Omron Sysmac Studio project TicTacToe (Sysmac Studio 1.60.0.64010, StandardProject)

# Controller new_Controller_0: NJ501-1500 version 1.67
Units and slaves: Power Supply : NJ-Px3001; CPU : NJ501-1500
Task PrimaryTask (priority 4, period or condition 1000): Program0

VAR_GLOBAL CONSTANT
    Table_HMI_Mapping : ARRAY[0..2,0..2] of uint := [1, 2, 3, 4, 5, 6, 7, 8, 9];  (* Use for HMI input mapping ONYL *)
END_VAR
VAR_GLOBAL
    Game_Start : BOOL;  (* Game Start Indicator *)
    Game_ReStart : BOOL;  (* Restart BTN *)
    PlayTable : ARRAY[0..2,0..2] of uint := [9(0)];
    Game_End : BOOL;  (* Game End Indicator *)
    WINNING_PLAYER : UINT;
    Player_Click : BOOL;  (* HMI BTN Detected *)
    BTN_LOCATION : UINT;
    PLAYER_1_ON : BOOL;
    PLAYER_2_ON : BOOL;
    row : UINT;
    col : UINT;
END_VAR

PROGRAM Program0
VAR
    CLEAR_TABLE : BOOL;  (* CLEAR TABLE DATA *)
    PLAYER_1_ACTIVATE : BOOL;
    PLAYER_2_ACTIVATE : BOOL;
    SWITCH_PLAYER : BOOL;
    INST_VALUE : UINT;  (* 0 = ERROR /       1= PLAYER_1        2= PLAYER_2 *)
    CheckInput : BOOL;
    CheckInput_DONE : BOOL;
END_VAR
VAR CONSTANT
    Table_Mapping_Col : Array[0..9] of Uint := [5, 0, 1, 2, 0, 1, 2, 0, 1, 2];
    Table_Mapping_Row : Array[0..9] of Uint := [5, 3(0), 3(1), 3(2)];
END_VAR
VAR_EXTERNAL
    Game_Start : BOOL;
    Game_ReStart : BOOL;
    PlayTable : ARRAY[0..2,0..2] of uint;
    Game_End : BOOL;
    WINNING_PLAYER : UINT;
    Player_Click : BOOL;
    PLAYER_1_ON : BOOL;
    PLAYER_2_ON : BOOL;
    BTN_LOCATION : UINT;
    row : UINT;
    col : UINT;
END_VAR
VAR
    _p1 : BOOL;
    _e2 : R_TRIG;
    _p3 : BOOL;
    _e4 : R_TRIG;
    _p5 : BOOL;
    _p6 : BOOL;
    _p7 : BOOL;
    _e8 : R_TRIG;
    _e9 : R_TRIG;
    _e10 : R_TRIG;
    _p11 : BOOL;
    _e12 : R_TRIG;
    _e13 : R_TRIG;
    _e14 : R_TRIG;
    _p15 : BOOL;
    _e16 : R_TRIG;
    _e17 : R_TRIG;
    _e18 : R_TRIG;
    _p19 : BOOL;
    _e20 : R_TRIG;
    _e21 : R_TRIG;
    _e22 : R_TRIG;
    _p23 : BOOL;
    _e24 : R_TRIG;
    _e25 : R_TRIG;
    _e26 : R_TRIG;
    _p27 : BOOL;
    _e28 : R_TRIG;
    _e29 : R_TRIG;
    _e30 : R_TRIG;
    _p31 : BOOL;
    _e32 : R_TRIG;
    _e33 : R_TRIG;
    _e34 : R_TRIG;
    _p35 : BOOL;
    _e36 : R_TRIG;
    _e37 : R_TRIG;
    _e38 : R_TRIG;
    _p39 : BOOL;
END_VAR

(* Section Main: ladder, written here as Structured Text *)

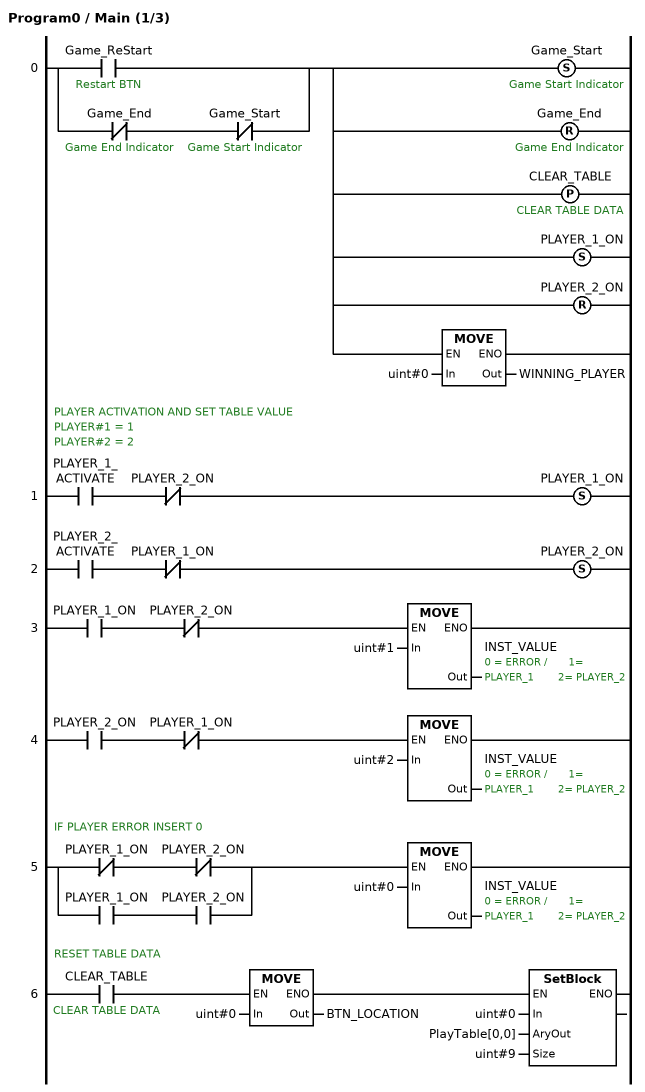
(* Rung 0 *)
_p1 := Game_ReStart OR (NOT Game_End AND NOT Game_Start);
IF _p1 THEN
    Game_Start := TRUE;
    Game_End := FALSE;
END_IF;
_e2(CLK := _p1);
CLEAR_TABLE := _e2.Q;
IF _p1 THEN
    PLAYER_1_ON := TRUE;
    PLAYER_2_ON := FALSE;
    WINNING_PLAYER := uint#0;
END_IF;
(* Rung 1: PLAYER ACTIVATION AND SET TABLE VALUE / PLAYER#1 = 1 / PLAYER#2 = 2 *)
IF PLAYER_1_ACTIVATE AND NOT PLAYER_2_ON THEN PLAYER_1_ON := TRUE; END_IF;
(* Rung 2 *)
IF PLAYER_2_ACTIVATE AND NOT PLAYER_1_ON THEN PLAYER_2_ON := TRUE; END_IF;
(* Rung 3 *)
IF PLAYER_1_ON AND NOT PLAYER_2_ON THEN INST_VALUE := uint#1; END_IF;
(* Rung 4 *)
IF PLAYER_2_ON AND NOT PLAYER_1_ON THEN INST_VALUE := uint#2; END_IF;
(* Rung 5: IF PLAYER ERROR INSERT 0 *)
IF (NOT PLAYER_1_ON AND NOT PLAYER_2_ON) OR (PLAYER_1_ON AND PLAYER_2_ON) THEN
    INST_VALUE := uint#0;
END_IF;
(* Rung 6: RESET TABLE DATA *)
IF CLEAR_TABLE THEN
    BTN_LOCATION := uint#0;
    SetBlock(In := uint#0, AryOut := PlayTable[0,0], Size := uint#9);
END_IF;

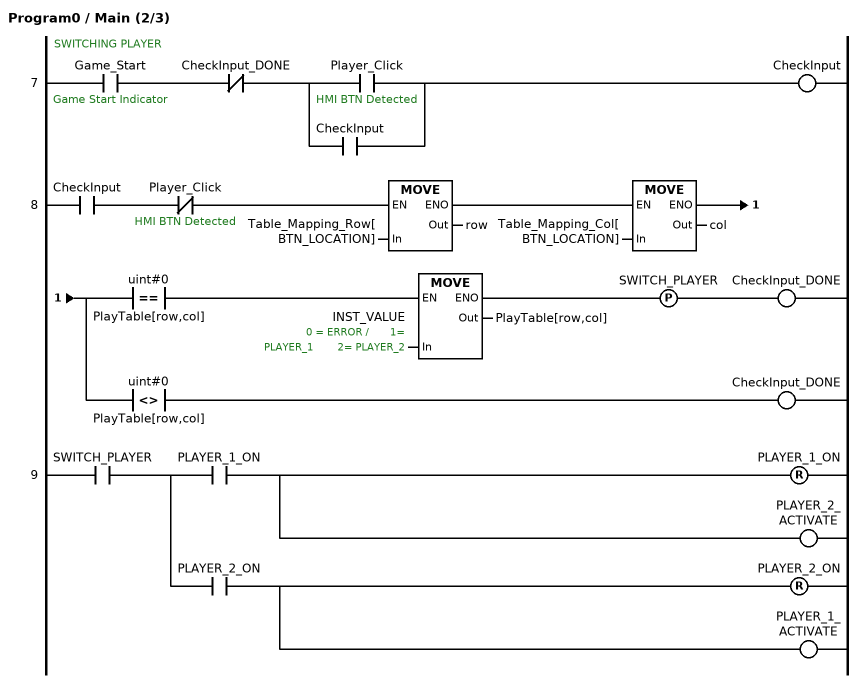
(* Rung 7: SWITCHING PLAYER *)
CheckInput := Game_Start AND NOT CheckInput_DONE AND (Player_Click OR CheckInput);
(* Rung 8 *)
IF CheckInput AND NOT Player_Click THEN
    row := Table_Mapping_Row[BTN_LOCATION];
    col := Table_Mapping_Col[BTN_LOCATION];
END_IF;
_p3 := CheckInput AND NOT Player_Click AND (uint#0 = PlayTable[row,col]);
IF _p3 THEN PlayTable[row,col] := INST_VALUE; END_IF;
_e4(CLK := _p3);
SWITCH_PLAYER := _e4.Q;
CheckInput_DONE := _p3;
CheckInput_DONE := CheckInput AND NOT Player_Click AND (uint#0 <> PlayTable[row,col]);
(* notes on elements: Check if the box is null *)
(* Rung 9 *)
_p5 := SWITCH_PLAYER AND PLAYER_1_ON;
IF _p5 THEN PLAYER_1_ON := FALSE; END_IF;
PLAYER_2_ACTIVATE := _p5;
_p6 := SWITCH_PLAYER AND PLAYER_2_ON;
IF _p6 THEN PLAYER_2_ON := FALSE; END_IF;
PLAYER_1_ACTIVATE := _p6;

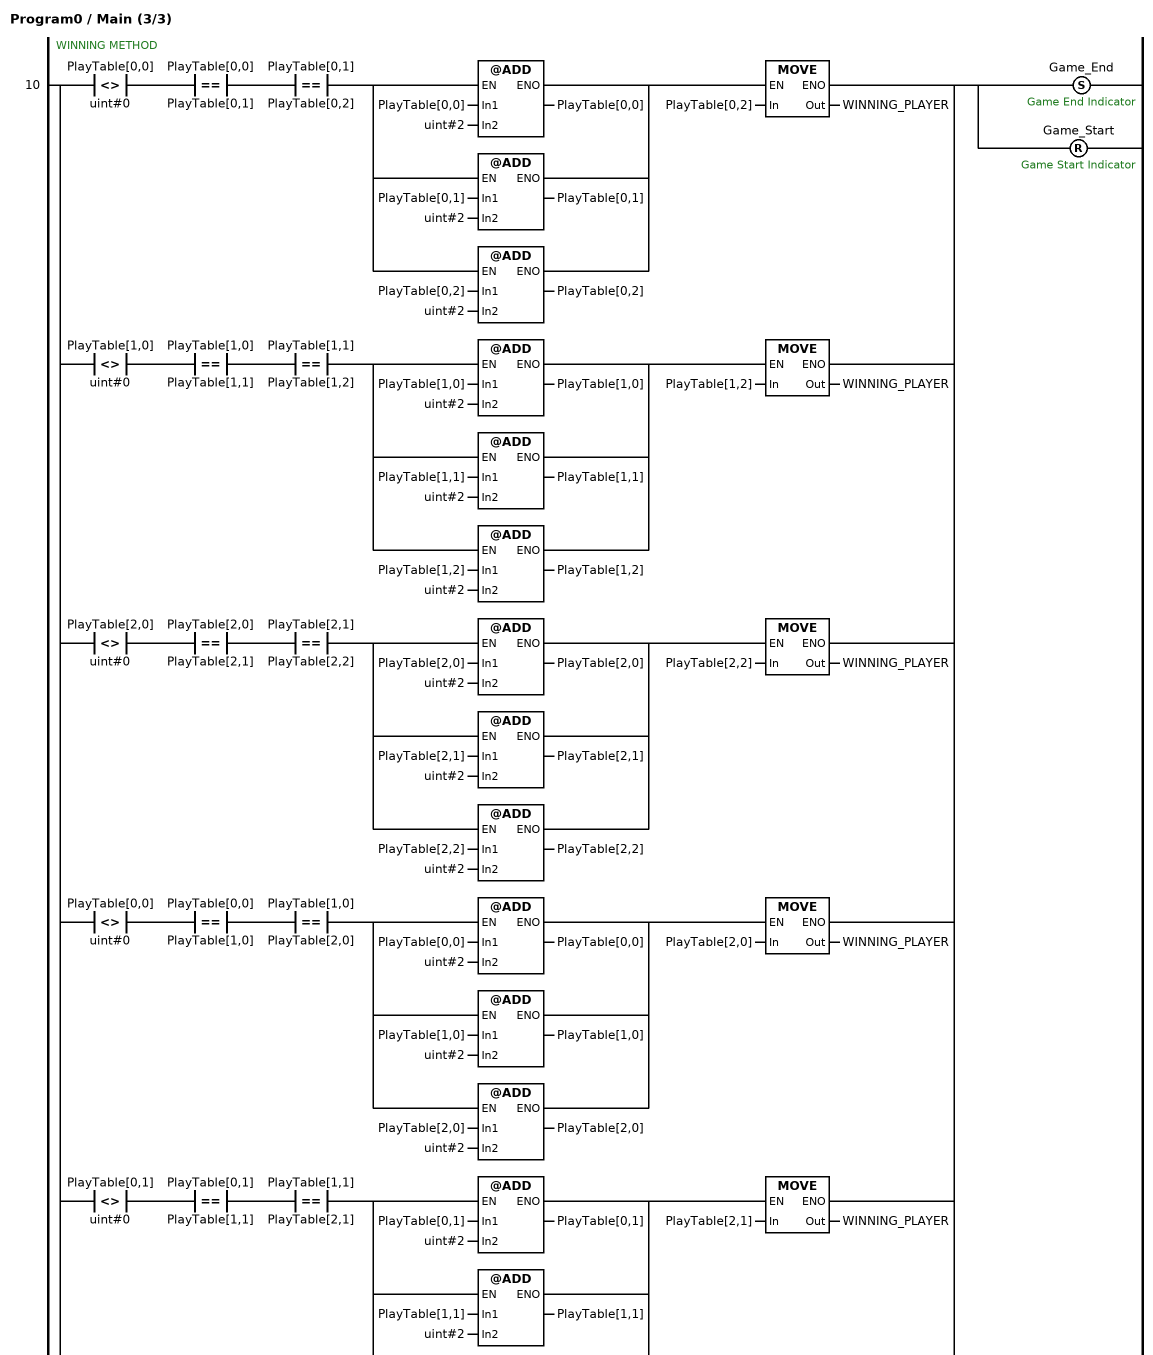

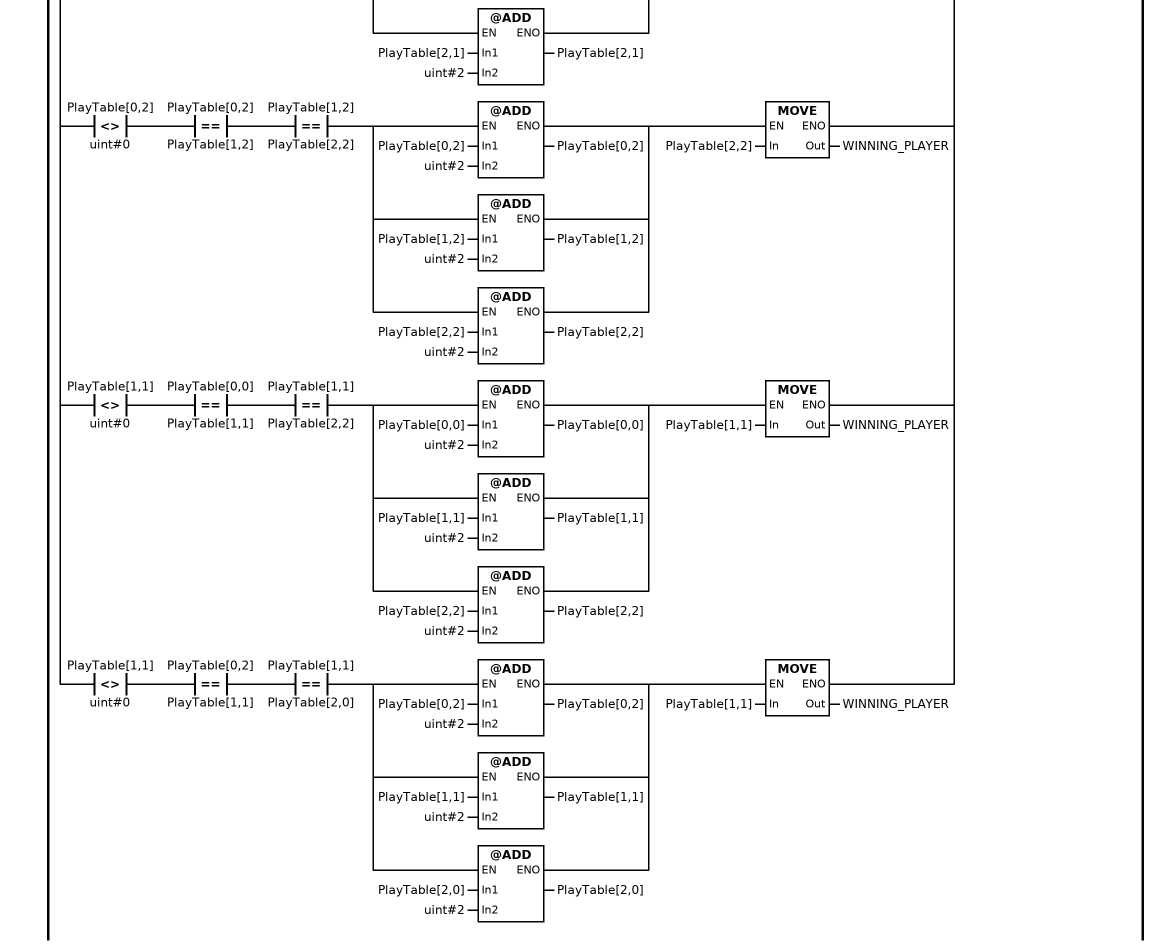
(* Rung 10: WINNING METHOD *)
_p7 := (PlayTable[0,0] <> uint#0) AND (PlayTable[0,0] = PlayTable[0,1]) AND (PlayTable[0,1] = PlayTable[0,2]);
_e8(CLK := _p7);
IF _e8.Q THEN PlayTable[0,0] := PlayTable[0,0] + uint#2; END_IF;
_e9(CLK := _p7);
IF _e9.Q THEN PlayTable[0,1] := PlayTable[0,1] + uint#2; END_IF;
_e10(CLK := _p7);
IF _e10.Q THEN PlayTable[0,2] := PlayTable[0,2] + uint#2; END_IF;
IF _e8.Q OR _e9.Q OR _e10.Q THEN WINNING_PLAYER := PlayTable[0,2]; END_IF;
_p11 := (PlayTable[1,0] <> uint#0) AND (PlayTable[1,0] = PlayTable[1,1]) AND (PlayTable[1,1] = PlayTable[1,2]);
_e12(CLK := _p11);
IF _e12.Q THEN PlayTable[1,0] := PlayTable[1,0] + uint#2; END_IF;
_e13(CLK := _p11);
IF _e13.Q THEN PlayTable[1,1] := PlayTable[1,1] + uint#2; END_IF;
_e14(CLK := _p11);
IF _e14.Q THEN PlayTable[1,2] := PlayTable[1,2] + uint#2; END_IF;
IF _e12.Q OR _e13.Q OR _e14.Q THEN WINNING_PLAYER := PlayTable[1,2]; END_IF;
_p15 := (PlayTable[2,0] <> uint#0) AND (PlayTable[2,0] = PlayTable[2,1]) AND (PlayTable[2,1] = PlayTable[2,2]);
_e16(CLK := _p15);
IF _e16.Q THEN PlayTable[2,0] := PlayTable[2,0] + uint#2; END_IF;
_e17(CLK := _p15);
IF _e17.Q THEN PlayTable[2,1] := PlayTable[2,1] + uint#2; END_IF;
_e18(CLK := _p15);
IF _e18.Q THEN PlayTable[2,2] := PlayTable[2,2] + uint#2; END_IF;
IF _e16.Q OR _e17.Q OR _e18.Q THEN WINNING_PLAYER := PlayTable[2,2]; END_IF;
_p19 := (PlayTable[0,0] <> uint#0) AND (PlayTable[0,0] = PlayTable[1,0]) AND (PlayTable[1,0] = PlayTable[2,0]);
_e20(CLK := _p19);
IF _e20.Q THEN PlayTable[0,0] := PlayTable[0,0] + uint#2; END_IF;
_e21(CLK := _p19);
IF _e21.Q THEN PlayTable[1,0] := PlayTable[1,0] + uint#2; END_IF;
_e22(CLK := _p19);
IF _e22.Q THEN PlayTable[2,0] := PlayTable[2,0] + uint#2; END_IF;
IF _e20.Q OR _e21.Q OR _e22.Q THEN WINNING_PLAYER := PlayTable[2,0]; END_IF;
_p23 := (PlayTable[0,1] <> uint#0) AND (PlayTable[0,1] = PlayTable[1,1]) AND (PlayTable[1,1] = PlayTable[2,1]);
_e24(CLK := _p23);
IF _e24.Q THEN PlayTable[0,1] := PlayTable[0,1] + uint#2; END_IF;
_e25(CLK := _p23);
IF _e25.Q THEN PlayTable[1,1] := PlayTable[1,1] + uint#2; END_IF;
_e26(CLK := _p23);
IF _e26.Q THEN PlayTable[2,1] := PlayTable[2,1] + uint#2; END_IF;
IF _e24.Q OR _e25.Q OR _e26.Q THEN WINNING_PLAYER := PlayTable[2,1]; END_IF;
_p27 := (PlayTable[0,2] <> uint#0) AND (PlayTable[0,2] = PlayTable[1,2]) AND (PlayTable[1,2] = PlayTable[2,2]);
_e28(CLK := _p27);
IF _e28.Q THEN PlayTable[0,2] := PlayTable[0,2] + uint#2; END_IF;
_e29(CLK := _p27);
IF _e29.Q THEN PlayTable[1,2] := PlayTable[1,2] + uint#2; END_IF;
_e30(CLK := _p27);
IF _e30.Q THEN PlayTable[2,2] := PlayTable[2,2] + uint#2; END_IF;
IF _e28.Q OR _e29.Q OR _e30.Q THEN WINNING_PLAYER := PlayTable[2,2]; END_IF;
_p31 := (PlayTable[1,1] <> uint#0) AND (PlayTable[0,0] = PlayTable[1,1]) AND (PlayTable[1,1] = PlayTable[2,2]);
_e32(CLK := _p31);
IF _e32.Q THEN PlayTable[0,0] := PlayTable[0,0] + uint#2; END_IF;
_e33(CLK := _p31);
IF _e33.Q THEN PlayTable[1,1] := PlayTable[1,1] + uint#2; END_IF;
_e34(CLK := _p31);
IF _e34.Q THEN PlayTable[2,2] := PlayTable[2,2] + uint#2; END_IF;
IF _e32.Q OR _e33.Q OR _e34.Q THEN WINNING_PLAYER := PlayTable[1,1]; END_IF;
_p35 := (PlayTable[1,1] <> uint#0) AND (PlayTable[0,2] = PlayTable[1,1]) AND (PlayTable[1,1] = PlayTable[2,0]);
_e36(CLK := _p35);
IF _e36.Q THEN PlayTable[0,2] := PlayTable[0,2] + uint#2; END_IF;
_e37(CLK := _p35);
IF _e37.Q THEN PlayTable[1,1] := PlayTable[1,1] + uint#2; END_IF;
_e38(CLK := _p35);
IF _e38.Q THEN PlayTable[2,0] := PlayTable[2,0] + uint#2; END_IF;
IF _e36.Q OR _e37.Q OR _e38.Q THEN WINNING_PLAYER := PlayTable[1,1]; END_IF;
_p39 := _e8.Q OR _e9.Q OR _e10.Q OR _e12.Q OR _e13.Q OR _e14.Q OR _e16.Q OR _e17.Q OR _e18.Q OR _e20.Q OR _e21.Q OR _e22.Q OR _e24.Q OR _e25.Q OR _e26.Q OR _e28.Q OR _e29.Q OR _e30.Q OR _e32.Q OR _e33.Q OR _e34.Q OR _e36.Q OR _e37.Q OR _e38.Q;
IF _p39 THEN
    Game_End := TRUE;
    Game_Start := FALSE;
END_IF;
(* notes on elements: ROW#1 WON; ROW#2 WON; ROW#3 WON; COL#1 WON; COL#2 WON; COL#3 WON; DIAG#1 WON; DIAG#2 WON *)
END_PROGRAM

# Device HMI_NA5_0 (NA): not converted